{attribute 'GeneratedUsingTerminal: EL3403-0000-0017'}
{attribute addProperty BoxType "EL3403-0000-0017"}
{attribute addProperty Id "Sync_ErrorAT %I*BOOL1TxPDO_ToggleAT %I*BOOL1CurrentAT %I*DINT4VoltageAT %I*DINT4Active_powerAT %I*DINT4IndexAT %I*USINT1VariantValueAT %I*DINT4"}
{attribute addProperty CRC "1762251782"}
{attribute addProperty Size "19"}
TYPE PM_Inputs_Channel_6909D406 :
STRUCT
	{attribute addProperty Name "Sync_Error"}
	Sync_Error AT %I* : BOOL;
	{attribute addProperty Name "TxPDO_Toggle"}
	TxPDO_Toggle AT %I* : BOOL;
	{attribute addProperty Name "Current"}
	Current AT %I* : DINT;
	{attribute addProperty Name "Voltage"}
	Voltage AT %I* : DINT;
	{attribute addProperty Name "Active_power"}
	Active_power AT %I* : DINT;
	{attribute addProperty Name "Index"}
	Index AT %I* : USINT;
	{attribute addProperty Name "VariantValue"}
	VariantValue AT %I* : DINT;
END_STRUCT
END_TYPE

(* stored: Version 1.2.0.0, ProductVersion 3.1.4024.9
   DUT PM_Inputs_Channel_6909D406: Id {0d7c0295-b07f-42ab-b0ba-6f26fad42eab} *)
